SUBAPPLICATION Uebung_055 (* DigitalInput_I1 auf DigitalOutput_Q1 *)
  (* Standard: 61499-2 *)
  (* Version 1.0, 2023-10-23, franz *)
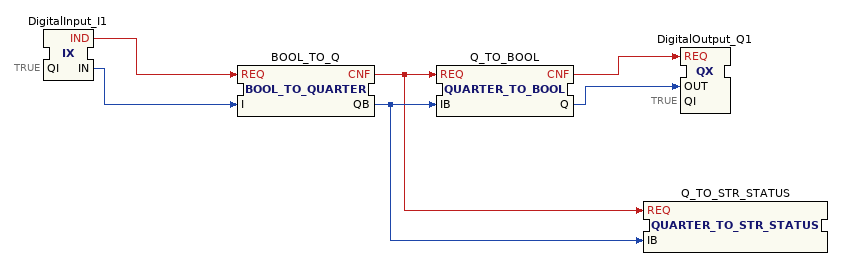
  FBS
    DigitalOutput_Q1 : QX(QI := TRUE);
    DigitalInput_I1 : IX(QI := TRUE);
    Q_TO_STR_STATUS : QUARTER_TO_STR_STATUS;
    Q_TO_BOOL : QUARTER_TO_BOOL;
    BOOL_TO_Q : BOOL_TO_QUARTER;
  END_FBS
  EVENT_CONNECTIONS
    Q_TO_BOOL.CNF TO DigitalOutput_Q1.REQ;
    DigitalInput_I1.IND TO BOOL_TO_Q.REQ;
    BOOL_TO_Q.CNF TO Q_TO_STR_STATUS.REQ;
    BOOL_TO_Q.CNF TO Q_TO_BOOL.REQ;
  END_CONNECTIONS
  DATA_CONNECTIONS
    Q_TO_BOOL.Q TO DigitalOutput_Q1.OUT;
    DigitalInput_I1.IN TO BOOL_TO_Q.I;
    BOOL_TO_Q.QB TO Q_TO_STR_STATUS.IB;
    BOOL_TO_Q.QB TO Q_TO_BOOL.IB;
  END_CONNECTIONS
END_SUBAPPLICATION
